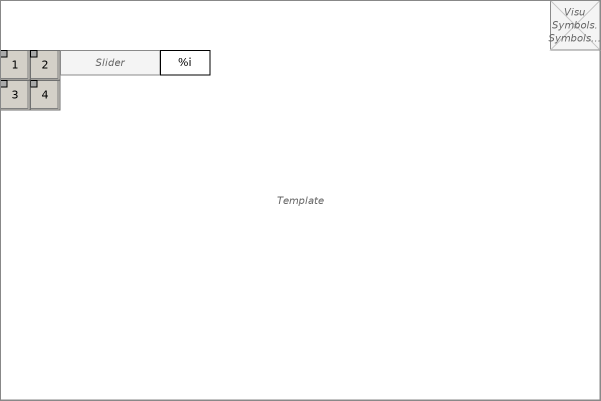
VISUALIZATION V_Hall  // 601x401
    Frame (0,0 601x401)
        shows Template()
    Image (550,0 50x50), image: VisuSymbols.Symbols.Home
        OnMouseClick: change screen: V_House
    Button (0,50 30x30), "1"
        tap PRG_SmartHome.fbRoom.fbLamp[0].Key
    Rectangle (0,50 7x7), colour toggle: PRG_SmartHome.fbRoom.fbLamp[0].Lamp
    Button (30,50 30x30), "2"
        tap PRG_SmartHome.fbRoom.fbLamp[1].Key
    Rectangle (30,50 7x7), colour toggle: PRG_SmartHome.fbRoom.fbLamp[1].Lamp
    Button (30,80 30x30), "4"
        tap PRG_SmartHome.fbRoom.fbLamp[3].Key
    Rectangle (30,80 7x7), colour toggle: PRG_SmartHome.fbRoom.fbLamp[3].Lamp
    Button (0,80 30x30), "3"
        tap PRG_SmartHome.fbRoom.fbLamp[2].Key
    Rectangle (0,80 7x7), colour toggle: PRG_SmartHome.fbRoom.fbLamp[2].Lamp
    Slider (60,50 100x25), variable: PRG_SmartHome.fbRoom.fbDimmer[0].rotarySw, scale 0..100
    Rectangle (160,50 50x25), "%i", text variable: PRG_SmartHome.fbRoom.fbDimmer[0].Dimmer
END_VISUALIZATION

(* stored: Version 1.1.0.1, ProductVersion 3.1.4024.12
   Visu V_Hall: Id {3ca749b6-3f9a-4690-bcec-90dae3dd78d0} *)
